(* Logix 5000 project; controller Planta_de_Kumis vendor 1 type 14 code 54 rev 20.11; software revision 20.00 *)

TASK Mapeo_IO (periodic, rate 10 ms, priority 6, watchdog 500 ms) : Mapeo_CadSim_Plus
TASK Rutina (periodic, rate 50 ms, priority 8, watchdog 500 ms) : MainProgram

MODULES
   Local : vendor 1 type 14 code 54 (ICP 0, rev 20.11)
END_MODULES

VAR_GLOBAL   (* controller tags *)
   Azucar : BOOL;
   Cultivo : BOOL;
   CV_TCV_201_1 : REAL;
   CV_TCV_202_1 : REAL;
   FI_01 : REAL;   // Indicador de flujo del vapor Intercambiador 1
   FI_02 : REAL;   // Indicador de flujo del agua Intercambiador 2
   FT_1 : REAL;
   HV1 : REAL;   // Valvula de entrada TK1
   HV2 : REAL;   // Valvula de desfogue
   HV3 : REAL;   // Valvula de desfogue TK2
   HV4 : REAL;   // Valvula de desfogue TK3
   HV5 : REAL;   // Valvula de desfogue TK4
   HV6 : REAL;   // Valvula de desfogue TK5
   HV7 : REAL;   // Valvula de desfogue TK6
   HV8 : REAL;   // Valvula de desfogue TK7
   HV9 : REAL;   // Valvula de desfogue TK8
   JY_01 : BOOL;   // Motor de mezclado M1
   JY_02 : BOOL;   // Motor de mezclado cultivo
   Leve_TK1 : REAL;   // Sensor de nivel TK1
   Level_TK10 : REAL;   // Sensor de nivel TK10 Intercambiador 2
   Level_TK2 : REAL;   // Sensor de nivel TK2
   Level_TK3 : REAL;   // Sensor de nivel TK·
   Level_TK4 : REAL;   // Sensor de nivel TK4
   Level_TK5 : REAL;   // Sensor de nivel TK5
   Level_TK6 : REAL;   // Sensor de nivel TK6
   Level_TK7 : REAL;   // Sensor de nivel TK7
   Level_TK8 : REAL;   // Sensor de nivel TK8
   Level_TK9 : REAL;   // Sensor de nivel TK9 Intercambiador 1
   LSH_101_1 : BOOL;   // Sensor de nivel alto TK1
   LSH_102_1 : BOOL;   // Sensor de nivel alto TK2
   LSH_103_1 : BOOL;   // Sensor de nivel alto TK3
   LSH_104_1 : BOOL;   // Sensor de nivel alto TK4
   LSH_105_1 : BOOL;   // Sensor de nivel alto TK5
   LSH_106_1 : BOOL;   // Sensor de nivel alto TK6
   LSH_107_1 : BOOL;   // Sensor de nivel alto TK7
   LSH_108_1 : BOOL;   // Sensor de nivel alto TK8
   LSL_101_1 : BOOL;   // Sensor de nivel bajo TK1
   LSL_102_1 : BOOL;   // Sensor de nivel bajo TK2
   LSL_103_1 : BOOL;   // Sensor de nivel bajo TK3
   LSL_104_1 : BOOL;   // Sensor de nivel bajo TK4
   LSL_105_1 : BOOL;   // Sensor de nivel bajo TK5
   LSL_106_1 : BOOL;   // Sensor de nivel bajo TK6
   LSL_107_1 : BOOL;   // Sensor de nivel baj TK7
   LSL_108_1 : BOOL;   // Sensor de nivel bajo TK8
   PI_01 : REAL;   // Indicador de presion del vapor Intercambiador 1
   PI_02 : REAL;   // Indicador de presion del agua Intercambiador 2
   PP1 : BOOL;   // Motobomba 1
   PP2 : BOOL;   // Motobomba 2
   PP3 : BOOL;   // Motobomba 3
   PP4 : BOOL;   // Motobomba 4
   PP5 : BOOL;   // Motobomba 5
   Start : BOOL;   // Boton de Inicio
   SV_101_1 : REAL;   // Valvula de salida TK1
   SV_102_1 : REAL;   // Valvula de salida TK2
   SV_103_1 : REAL;   // Valvula de salida TK3
   SV_104_1 : REAL;   // Valvula de salida
   SV_105_1 : REAL;   // Valvula de entrada TK5
   SV_106_1 : REAL;   // Valvula de entrada TK6
   SV_107_1 : REAL;   // Valvula de entrada TK7
   SV_108_1 : REAL;   // Valvula de entrada TK8
   SV_201_1 : REAL;   // Valvula de salida 1 Intercambiador
   SV_201_2 : REAL;   // Valvula de reflujo Intercambiador 1
   SV_202_1 : REAL;   // Valvula de salida 1 Intercambiador 2
   SV_202_2 : REAL;   // Valvula de reflujo
   T_Agua : DINT;   // Temperatura de entrada del Agua Fria
   T_Int : DINT;   // Temperatura de entrada de la leche
   TCV_101_1 : REAL;   // valvula de entrada al tanque de recepcion
   TCV_201_1 : REAL;   // Valvula de entrada de Vapor Variable manipulada
   TCV_202_1 : REAL;   // Valvula de entrada de agua Variable manipulada Intercambiador 2
   TI_01 : REAL;   // Indicador de temperatura TK1
   TI_02 : REAL;   // Indicador de temperatura TK2
   TI_03 : REAL;   // Indicador de temperatura del vapor Intercambiador 1
   TI_05 : REAL;   // Indicador de temperatura TK3
   TI_06 : REAL;   // Indicador de temperatura del agua
   TITE_201_1 : REAL := 60.726944;   // Sensor de temperatura de producto intermedio Variable Controlada Intercambiador 1
   TITE_202_1 : REAL := 42.013607;   // Sensor de temperatura de producto intermedio Variable controlada Intercambiador 2
   TITE_Prueba : REAL := 60.724613;
   TITE_Prueba_2 : REAL := 42.011265;
END_VAR

PROGRAM MainProgram   (* main routine MainRoutine *)
VAR
   BIT_MEZC_AZUCAR : BOOL;   // Indicador de mezclado de azucar
   BIT_MEZC_CULTIVO : BOOL;   // Bit indicador mezclado de cultivo
   BIT_PRUEBA : BOOL;
   BIT_PRUEBA_2 : BOOL;
   C1 : COUNTER := (PRE := 5);
   Latch_Azcuar_On : BOOL;
   Latch_LSH_TK1 : BOOL;
   Latch_LSH_TK2 : BOOL;
   Latch_LSH_TK3 : BOOL;
   Latch_LSH_TK4 : BOOL;
   Latch_LSH_TK5 : BOOL;
   Latch_LSH_TK6 : BOOL;
   Latch_LSH_TK7 : BOOL;
   Latch_LSH_TK8 : BOOL;
   Latch_OSR_2 : BOOL;
   Latch_OSR_4 : BOOL;
   Latch_OSR_6 : BOOL;
   Latch_OSR_8 : BOOL;
   Latch_SR1 : BOOL;
   Latch_SR2 : BOOL;
   Latch_Timer_Mezclado_DN : BOOL;
   Next_Batch : BOOL;
   OSR_1 : BOOL;
   OSR_2 : BOOL;
   OSR_3 : BOOL;
   OSR_4 : BOOL;
   OSR_5 : BOOL;
   OSR_6 : BOOL;
   OSR_7 : BOOL;
   OSR_8 : BOOL;
   PID_Exchanger_1 : PID := (CTL := 8397952, PE := 1, OLL := 1, DVNA := 1, PVHA := 1, SP := 60.0, KP := 0.029, KI := 61.247, KD := 15.352, MAXS := 100.0, MAXO := 100.0, UPD := 1.0, PV := 60.726944, ERR := -0.72694397, MAXI := 100.0, MAXCV := 100.0, DATA[0] := -0.008097162, DATA[1] := -23.727255, DATA[2] := 60.726944, DATA[3] := -0.72694397, DATA[4] := 60.0, DATA[5] := 0.024420025, DATA[6] := 1.0, DATA[7] := 2.6, DATA[8] := 11.0, DATA[9] := 2.95, DATA[10] := 1.0, DATA[11] := 11.0, DATA[12] := 2.95, DATA[13] := 1.0, DATA[15] := 1.0, DATA[16] := 1.0);   // PID para el intercambiado de calor con vapor
   PID_Exchanger_2 : PID := (CTL := 41944192, CA := 1, PE := 1, DVNA := 1, PVHA := 1, SP := 60.0, KP := 0.013, KI := 71.98, KD := 17.99, MAXS := 100.0, MAXO := 100.0, UPD := 1.0, PV := 41.797935, ERR := -0.20206451, OUT := 4.3428845, MAXI := 100.0, MAXCV := 100.0, DATA[0] := 4.456376, DATA[1] := 16.331306, DATA[2] := 41.797935, DATA[3] := -0.20206451, DATA[4] := 42.0, DATA[5] := 0.024420025, DATA[6] := 1.0, DATA[7] := 1.6, DATA[8] := 23.0, DATA[9] := 2.0, DATA[11] := 23.0, DATA[12] := 2.0, DATA[15] := 1.0, DATA[16] := 0.024420025);   // PID para el intercambiador de disminucion de temperatura
   Salida_Prueba_1 : BOOL;
   Timer_Azucar : TIMER := (PRE := 1000);
   Timer_Cultivo : TIMER := (PRE := 1000);
   Timer_Disminucion_T : TIMER;
   timer_Elevado_T : TIMER;
   Timer_Inoculado : TIMER := (PRE := 6000);
   Timer_Mezclado : TIMER := (PRE := 1000);
   Timer_Recepcion : TIMER := (PRE := 1000);
   Timer_TK5 : TIMER := (PRE := 5000);
   Timer_TK6 : TIMER := (PRE := 5000);
   Timer_TK7 : TIMER := (PRE := 5000);
   Timer_TK8 : TIMER := (PRE := 5000);
END_VAR

ROUTINE MainRoutine   (* ladder *)
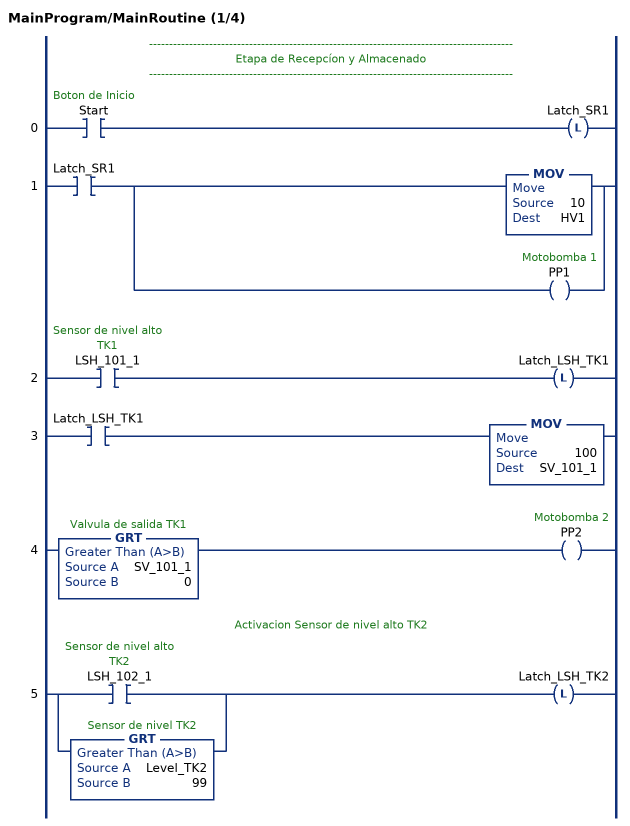
   // -------------------------------------------------------------------------------------------
   // Etapa de Recepcíon y Almacenado
   // -------------------------------------------------------------------------------------------
   0: XIC(Start)OTL(Latch_SR1);
   1: XIC(Latch_SR1)[MOV(10,HV1) ,OTE(PP1) ];
   2: XIC(LSH_101_1)OTL(Latch_LSH_TK1);
   3: XIC(Latch_LSH_TK1)MOV(100,SV_101_1);
   4: GRT(SV_101_1,0)OTE(PP2);
   // Activacion Sensor de nivel alto TK2
   5: [XIC(LSH_102_1) ,GRT(Level_TK2,99) ]OTL(Latch_LSH_TK2);
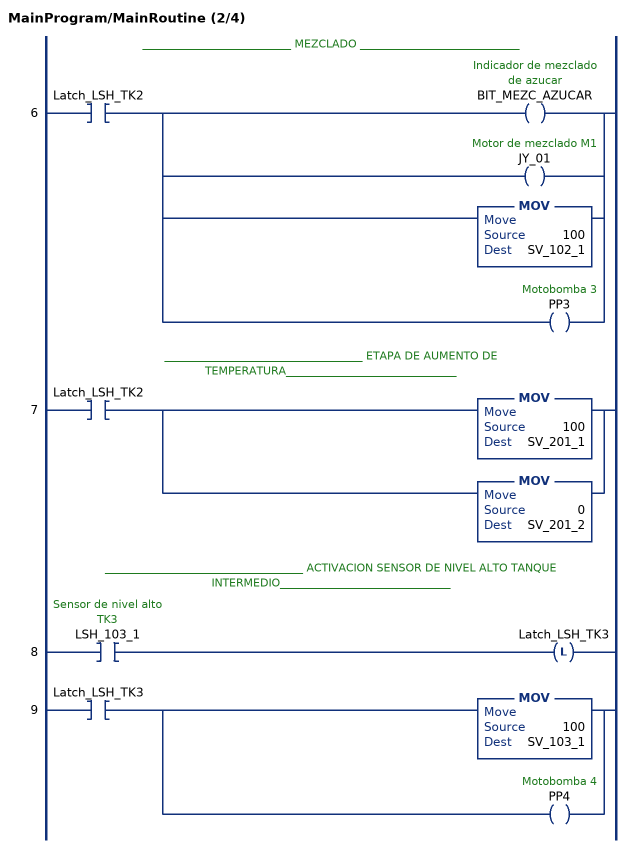
   // ___________________________ MEZCLADO _____________________________
   6: XIC(Latch_LSH_TK2)[OTE(BIT_MEZC_AZUCAR) ,[OTE(JY_01) ,[MOV(100,SV_102_1) ,OTE(PP3) ] ] ];
   // ____________________________________ ETAPA DE AUMENTO DE TEMPERATURA_______________________________
   7: XIC(Latch_LSH_TK2)[MOV(100,SV_201_1) ,MOV(0,SV_201_2) ];
   // ____________________________________ ACTIVACION SENSOR DE NIVEL ALTO TANQUE INTERMEDIO_______________________________
   8: XIC(LSH_103_1)OTL(Latch_LSH_TK3);
   9: XIC(Latch_LSH_TK3)[MOV(100,SV_103_1) ,OTE(PP4) ];
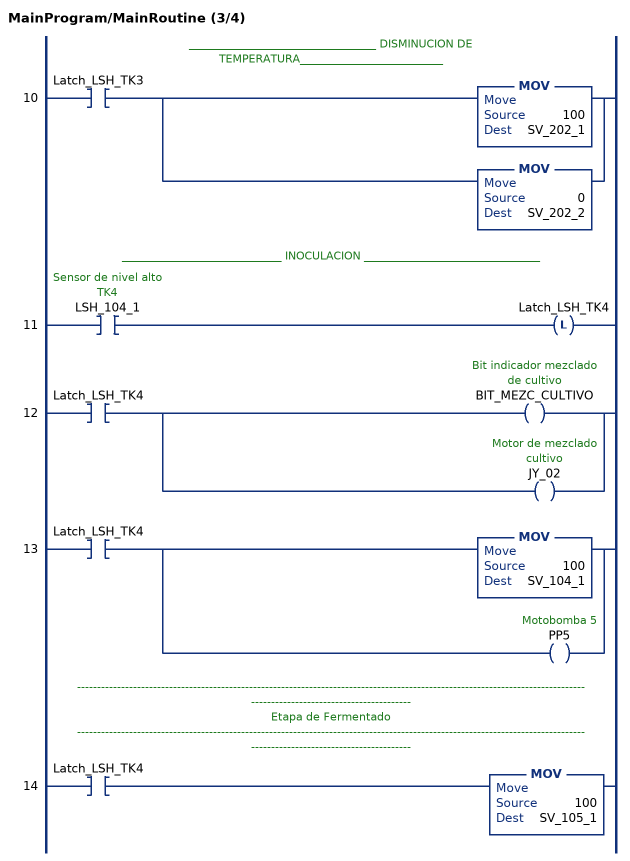
   // __________________________________ DISMINUCION DE TEMPERATURA__________________________
   10: XIC(Latch_LSH_TK3)[MOV(100,SV_202_1) ,MOV(0,SV_202_2) ];
   // _____________________________ INOCULACION ________________________________
   11: XIC(LSH_104_1)OTL(Latch_LSH_TK4);
   12: XIC(Latch_LSH_TK4)[OTE(BIT_MEZC_CULTIVO) ,OTE(JY_02) ];
   13: XIC(Latch_LSH_TK4)[MOV(100,SV_104_1) ,OTE(PP5) ];
   // -----------------------------------------------------------------------------------------------------------------------------------------------------------------------
   // Etapa de Fermentado
   // -----------------------------------------------------------------------------------------------------------------------------------------------------------------------
   14: XIC(Latch_LSH_TK4)MOV(100,SV_105_1);
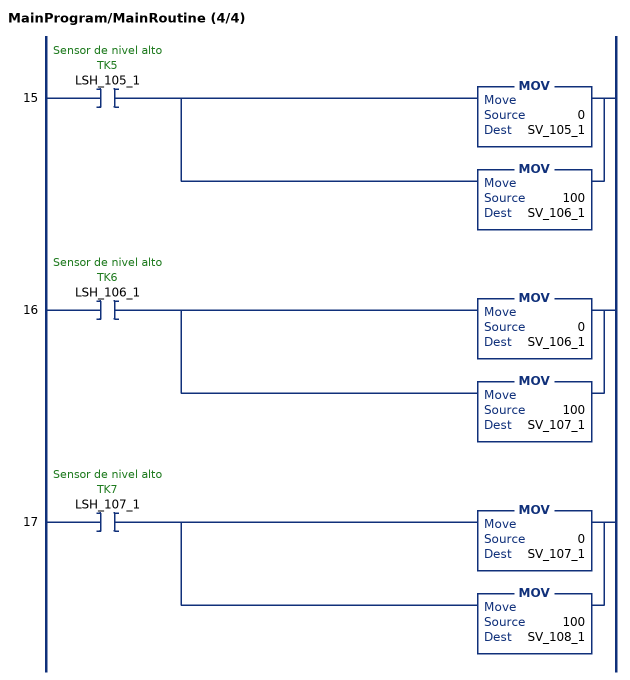
   15: XIC(LSH_105_1)[MOV(0,SV_105_1) ,MOV(100,SV_106_1) ];
   16: XIC(LSH_106_1)[MOV(0,SV_106_1) ,MOV(100,SV_107_1) ];
   17: XIC(LSH_107_1)[MOV(0,SV_107_1) ,MOV(100,SV_108_1) ];
END_ROUTINE
END_PROGRAM

PROGRAM Mapeo_CadSim_Plus   (* main routine Main *)

ROUTINE Main   (* ladder *)
END_ROUTINE

ROUTINE Mapeo1_DI   (* ladder *)
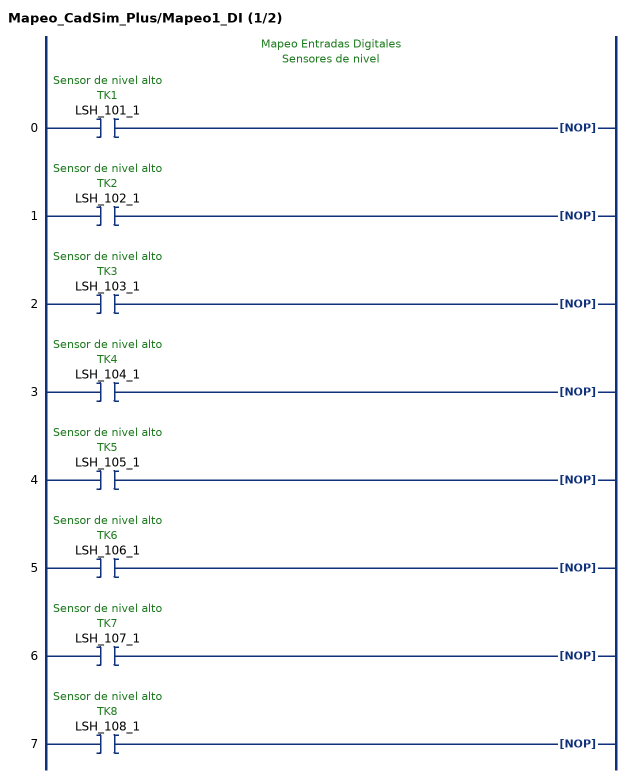
   // Mapeo Entradas Digitales
   // Sensores de nivel
   0: XIC(LSH_101_1)NOP();
   1: XIC(LSH_102_1)NOP();
   2: XIC(LSH_103_1)NOP();
   3: XIC(LSH_104_1)NOP();
   4: XIC(LSH_105_1)NOP();
   5: XIC(LSH_106_1)NOP();
   6: XIC(LSH_107_1)NOP();
   7: XIC(LSH_108_1)NOP();
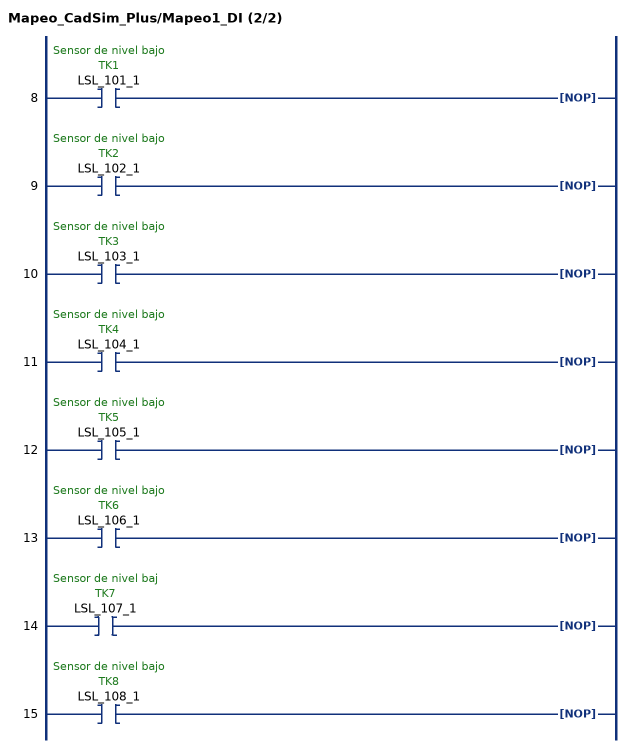
   8: XIC(LSL_101_1)NOP();
   9: XIC(LSL_102_1)NOP();
   10: XIC(LSL_103_1)NOP();
   11: XIC(LSL_104_1)NOP();
   12: XIC(LSL_105_1)NOP();
   13: XIC(LSL_106_1)NOP();
   14: XIC(LSL_107_1)NOP();
   15: XIC(LSL_108_1)NOP();
END_ROUTINE

ROUTINE Mapeo2_DO   (* ladder *)
END_ROUTINE

ROUTINE Mapeo3_AI   (* function block diagram *)
   SHEET 1
END_ROUTINE

ROUTINE Mapeo4_AO   (* ladder *)
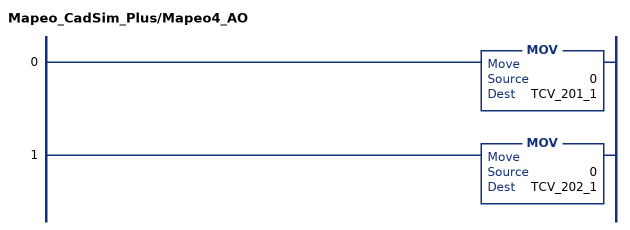
   0: MOV(0,TCV_201_1);
   1: MOV(0,TCV_202_1);
END_ROUTINE
END_PROGRAM
